FUNCTION_BLOCK Load
  (* Standard: 61499-2 *)
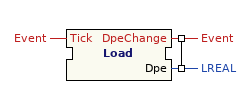
  EVENT_INPUT
    Tick;
  END_EVENT
  EVENT_OUTPUT
    DpeChange WITH Dpe;
  END_EVENT
  VAR_OUTPUT
    Dpe : LREAL;
  END_VAR
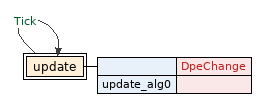
  EC_STATES
    update : -> DpeChange, update_alg0;
  END_STATES
  EC_TRANSITIONS
    update TO update := Tick;
  END_TRANSITIONS
  ALGORITHM update_alg0 IN ST:
Dpe := 0.20
  END_ALGORITHM
END_FUNCTION_BLOCK
